(* Logix 5000 project; controller BTS01 vendor 1 type 14 code 217 rev 32.14; software revision 32.04; part 6 of 15 *)
(* tags used below, declared in another part *)
   Alarm_Active : DINT;
   Alarm_TMR : TIMER[17,32];
   ALM_ENABLE : DINT[25];
   HMI_Global_Alarm_Ack_PB : BOOL;
   HMIAlarms : DINT[25];   // Alarm Trigger Array
   HMIAlarmsMsg : STRING64[17,32];   // Alarm Descriptions to Match Alarm Trigger Array
(* Alarm, continued *)

ROUTINE Alarm_04   (* ladder *)
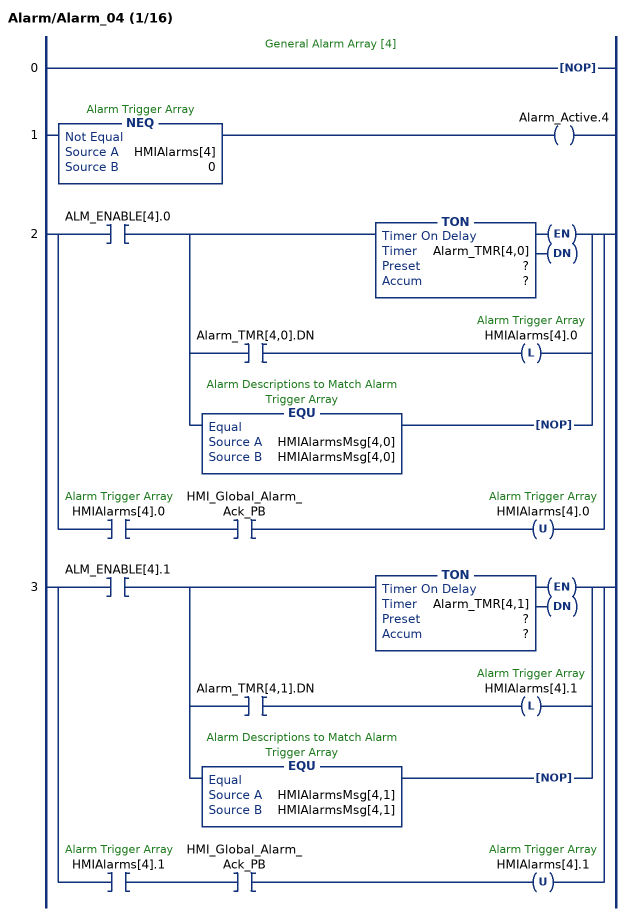
   // General Alarm Array [4]
   0: NOP();
   1: NEQ(HMIAlarms[4],0)OTE(Alarm_Active.4);
   2: [XIC(ALM_ENABLE[4].0) [TON(Alarm_TMR[4,0],?,?) ,XIC(Alarm_TMR[4,0].DN) OTL(HMIAlarms[4].0) ,EQU(HMIAlarmsMsg[4,0],HMIAlarmsMsg[4,0]) NOP() ] ,XIC(HMIAlarms[4].0) XIC(HMI_Global_Alarm_Ack_PB) OTU(HMIAlarms[4].0) ];
   3: [XIC(ALM_ENABLE[4].1) [TON(Alarm_TMR[4,1],?,?) ,XIC(Alarm_TMR[4,1].DN) OTL(HMIAlarms[4].1) ,EQU(HMIAlarmsMsg[4,1],HMIAlarmsMsg[4,1]) NOP() ] ,XIC(HMIAlarms[4].1) XIC(HMI_Global_Alarm_Ack_PB) OTU(HMIAlarms[4].1) ];
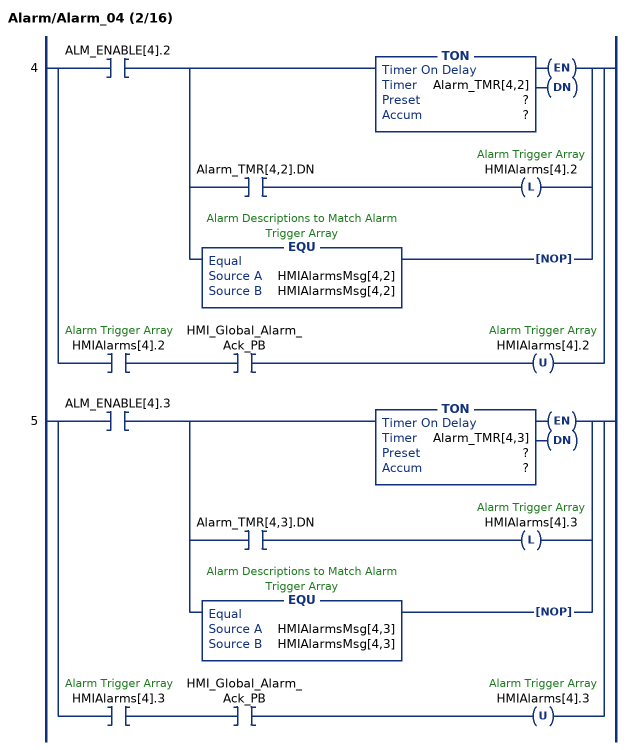
   4: [XIC(ALM_ENABLE[4].2) [TON(Alarm_TMR[4,2],?,?) ,XIC(Alarm_TMR[4,2].DN) OTL(HMIAlarms[4].2) ,EQU(HMIAlarmsMsg[4,2],HMIAlarmsMsg[4,2]) NOP() ] ,XIC(HMIAlarms[4].2) XIC(HMI_Global_Alarm_Ack_PB) OTU(HMIAlarms[4].2) ];
   5: [XIC(ALM_ENABLE[4].3) [TON(Alarm_TMR[4,3],?,?) ,XIC(Alarm_TMR[4,3].DN) OTL(HMIAlarms[4].3) ,EQU(HMIAlarmsMsg[4,3],HMIAlarmsMsg[4,3]) NOP() ] ,XIC(HMIAlarms[4].3) XIC(HMI_Global_Alarm_Ack_PB) OTU(HMIAlarms[4].3) ];
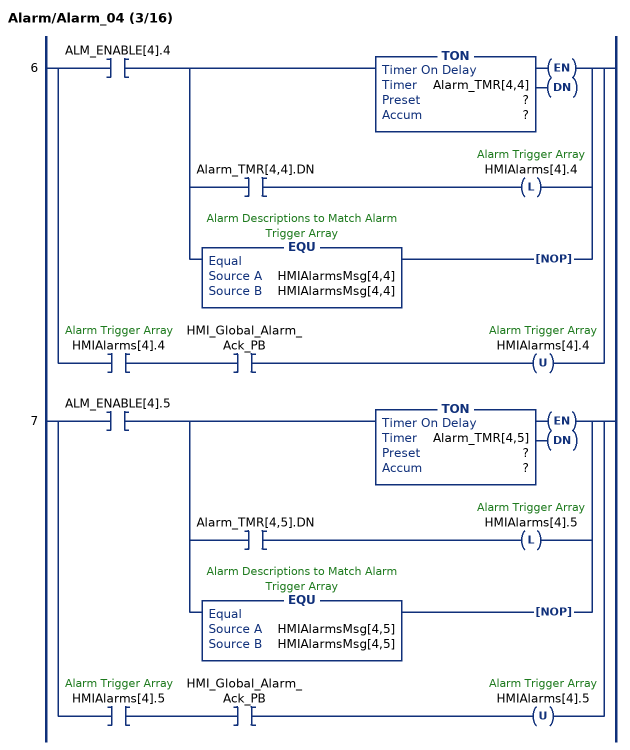
   6: [XIC(ALM_ENABLE[4].4) [TON(Alarm_TMR[4,4],?,?) ,XIC(Alarm_TMR[4,4].DN) OTL(HMIAlarms[4].4) ,EQU(HMIAlarmsMsg[4,4],HMIAlarmsMsg[4,4]) NOP() ] ,XIC(HMIAlarms[4].4) XIC(HMI_Global_Alarm_Ack_PB) OTU(HMIAlarms[4].4) ];
   7: [XIC(ALM_ENABLE[4].5) [TON(Alarm_TMR[4,5],?,?) ,XIC(Alarm_TMR[4,5].DN) OTL(HMIAlarms[4].5) ,EQU(HMIAlarmsMsg[4,5],HMIAlarmsMsg[4,5]) NOP() ] ,XIC(HMIAlarms[4].5) XIC(HMI_Global_Alarm_Ack_PB) OTU(HMIAlarms[4].5) ];
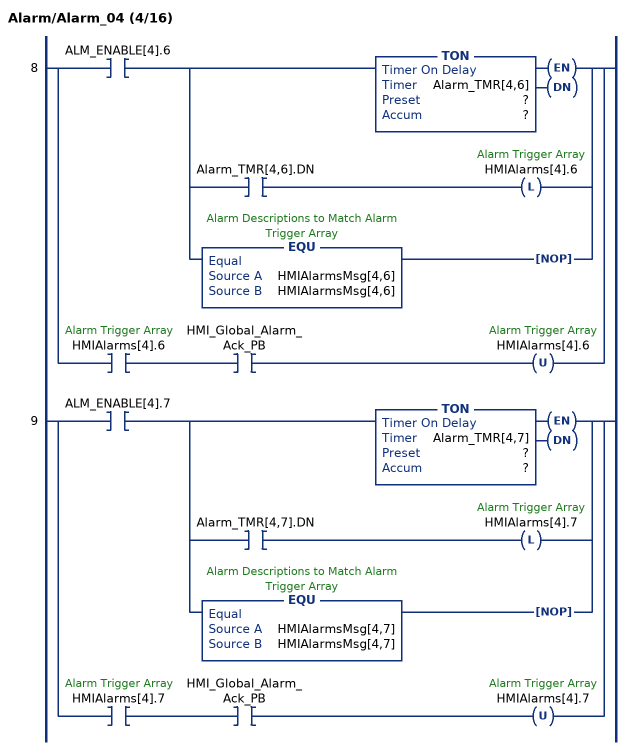
   8: [XIC(ALM_ENABLE[4].6) [TON(Alarm_TMR[4,6],?,?) ,XIC(Alarm_TMR[4,6].DN) OTL(HMIAlarms[4].6) ,EQU(HMIAlarmsMsg[4,6],HMIAlarmsMsg[4,6]) NOP() ] ,XIC(HMIAlarms[4].6) XIC(HMI_Global_Alarm_Ack_PB) OTU(HMIAlarms[4].6) ];
   9: [XIC(ALM_ENABLE[4].7) [TON(Alarm_TMR[4,7],?,?) ,XIC(Alarm_TMR[4,7].DN) OTL(HMIAlarms[4].7) ,EQU(HMIAlarmsMsg[4,7],HMIAlarmsMsg[4,7]) NOP() ] ,XIC(HMIAlarms[4].7) XIC(HMI_Global_Alarm_Ack_PB) OTU(HMIAlarms[4].7) ];
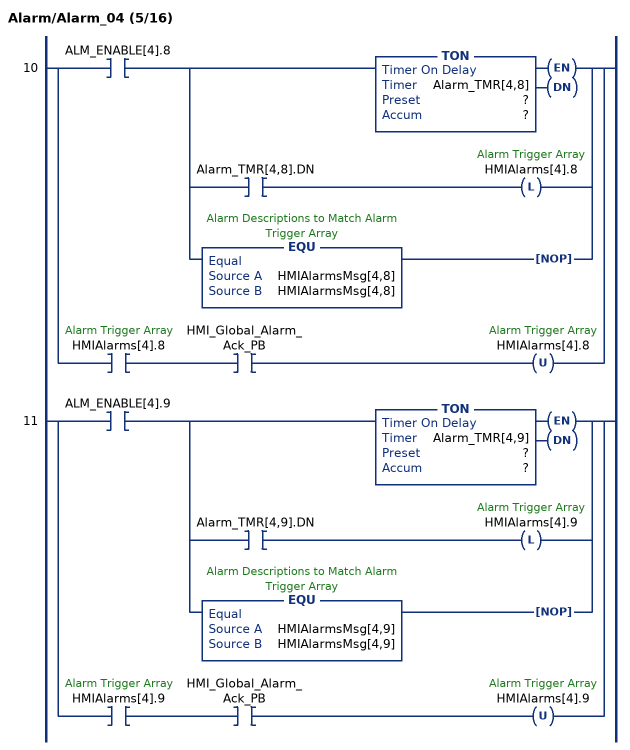
   10: [XIC(ALM_ENABLE[4].8) [TON(Alarm_TMR[4,8],?,?) ,XIC(Alarm_TMR[4,8].DN) OTL(HMIAlarms[4].8) ,EQU(HMIAlarmsMsg[4,8],HMIAlarmsMsg[4,8]) NOP() ] ,XIC(HMIAlarms[4].8) XIC(HMI_Global_Alarm_Ack_PB) OTU(HMIAlarms[4].8) ];
   11: [XIC(ALM_ENABLE[4].9) [TON(Alarm_TMR[4,9],?,?) ,XIC(Alarm_TMR[4,9].DN) OTL(HMIAlarms[4].9) ,EQU(HMIAlarmsMsg[4,9],HMIAlarmsMsg[4,9]) NOP() ] ,XIC(HMIAlarms[4].9) XIC(HMI_Global_Alarm_Ack_PB) OTU(HMIAlarms[4].9) ];
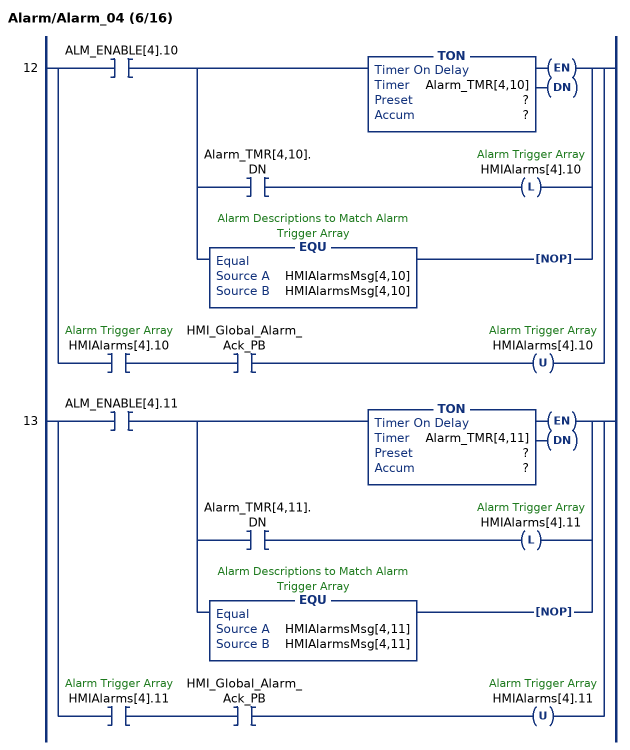
   12: [XIC(ALM_ENABLE[4].10) [TON(Alarm_TMR[4,10],?,?) ,XIC(Alarm_TMR[4,10].DN) OTL(HMIAlarms[4].10) ,EQU(HMIAlarmsMsg[4,10],HMIAlarmsMsg[4,10]) NOP() ] ,XIC(HMIAlarms[4].10) XIC(HMI_Global_Alarm_Ack_PB) OTU(HMIAlarms[4].10) ];
   13: [XIC(ALM_ENABLE[4].11) [TON(Alarm_TMR[4,11],?,?) ,XIC(Alarm_TMR[4,11].DN) OTL(HMIAlarms[4].11) ,EQU(HMIAlarmsMsg[4,11],HMIAlarmsMsg[4,11]) NOP() ] ,XIC(HMIAlarms[4].11) XIC(HMI_Global_Alarm_Ack_PB) OTU(HMIAlarms[4].11) ];
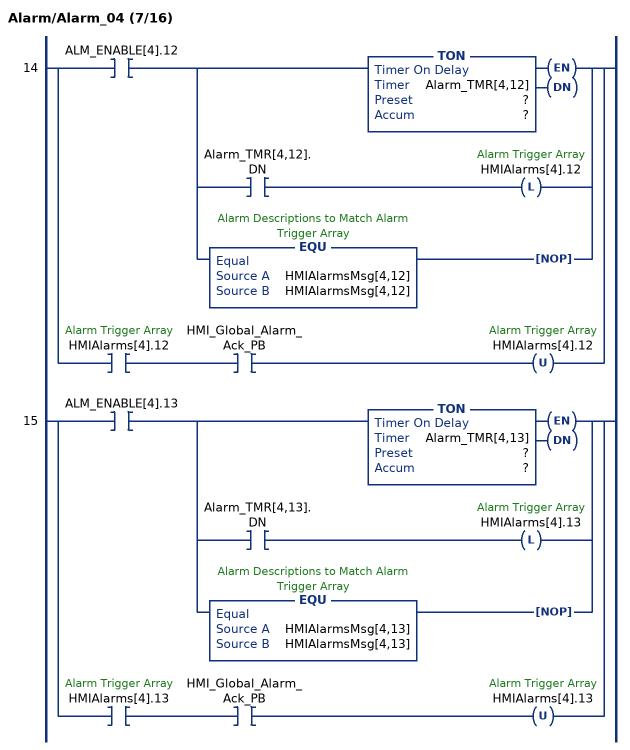
   14: [XIC(ALM_ENABLE[4].12) [TON(Alarm_TMR[4,12],?,?) ,XIC(Alarm_TMR[4,12].DN) OTL(HMIAlarms[4].12) ,EQU(HMIAlarmsMsg[4,12],HMIAlarmsMsg[4,12]) NOP() ] ,XIC(HMIAlarms[4].12) XIC(HMI_Global_Alarm_Ack_PB) OTU(HMIAlarms[4].12) ];
   15: [XIC(ALM_ENABLE[4].13) [TON(Alarm_TMR[4,13],?,?) ,XIC(Alarm_TMR[4,13].DN) OTL(HMIAlarms[4].13) ,EQU(HMIAlarmsMsg[4,13],HMIAlarmsMsg[4,13]) NOP() ] ,XIC(HMIAlarms[4].13) XIC(HMI_Global_Alarm_Ack_PB) OTU(HMIAlarms[4].13) ];
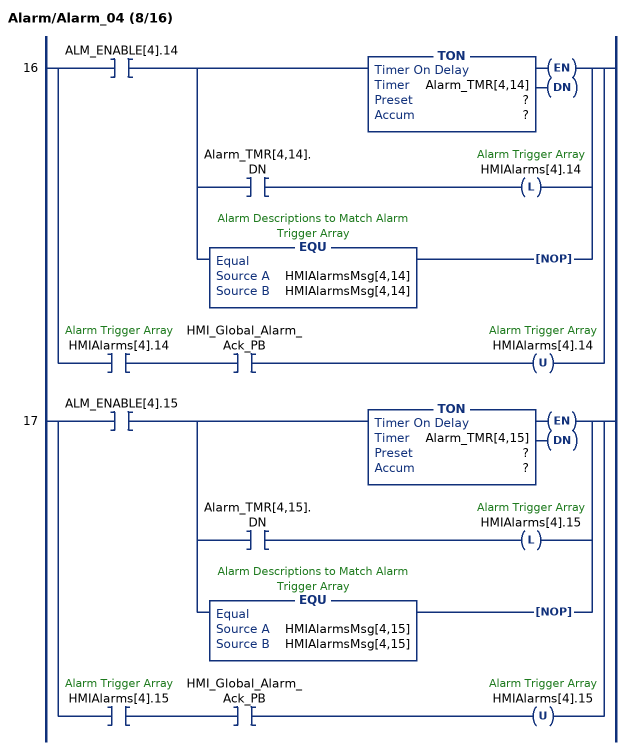
   16: [XIC(ALM_ENABLE[4].14) [TON(Alarm_TMR[4,14],?,?) ,XIC(Alarm_TMR[4,14].DN) OTL(HMIAlarms[4].14) ,EQU(HMIAlarmsMsg[4,14],HMIAlarmsMsg[4,14]) NOP() ] ,XIC(HMIAlarms[4].14) XIC(HMI_Global_Alarm_Ack_PB) OTU(HMIAlarms[4].14) ];
   17: [XIC(ALM_ENABLE[4].15) [TON(Alarm_TMR[4,15],?,?) ,XIC(Alarm_TMR[4,15].DN) OTL(HMIAlarms[4].15) ,EQU(HMIAlarmsMsg[4,15],HMIAlarmsMsg[4,15]) NOP() ] ,XIC(HMIAlarms[4].15) XIC(HMI_Global_Alarm_Ack_PB) OTU(HMIAlarms[4].15) ];
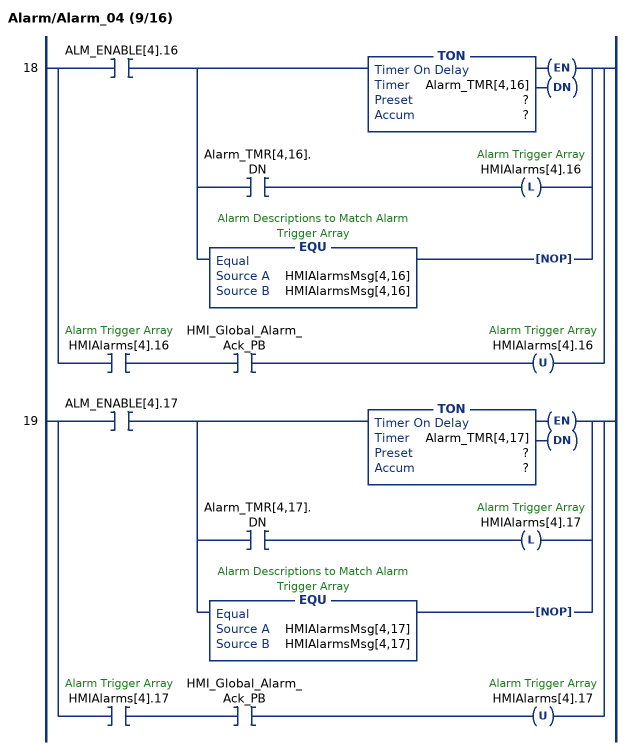
   18: [XIC(ALM_ENABLE[4].16) [TON(Alarm_TMR[4,16],?,?) ,XIC(Alarm_TMR[4,16].DN) OTL(HMIAlarms[4].16) ,EQU(HMIAlarmsMsg[4,16],HMIAlarmsMsg[4,16]) NOP() ] ,XIC(HMIAlarms[4].16) XIC(HMI_Global_Alarm_Ack_PB) OTU(HMIAlarms[4].16) ];
   19: [XIC(ALM_ENABLE[4].17) [TON(Alarm_TMR[4,17],?,?) ,XIC(Alarm_TMR[4,17].DN) OTL(HMIAlarms[4].17) ,EQU(HMIAlarmsMsg[4,17],HMIAlarmsMsg[4,17]) NOP() ] ,XIC(HMIAlarms[4].17) XIC(HMI_Global_Alarm_Ack_PB) OTU(HMIAlarms[4].17) ];
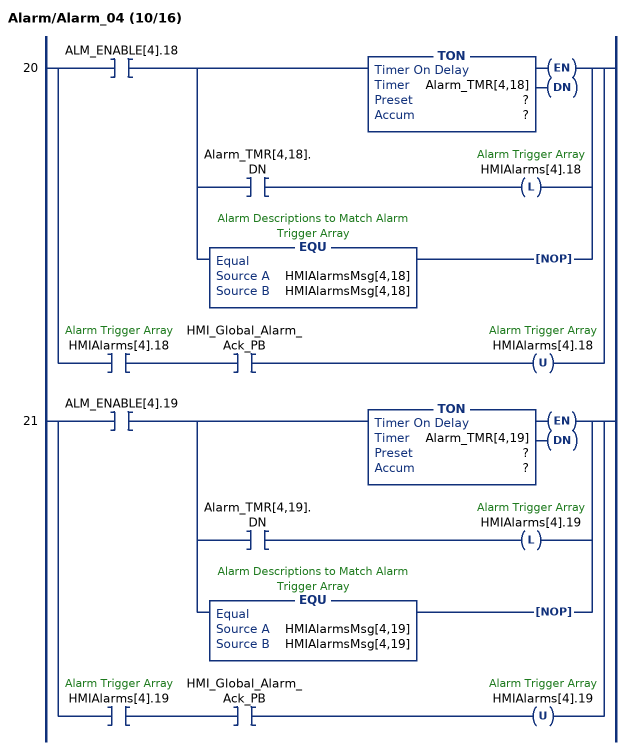
   20: [XIC(ALM_ENABLE[4].18) [TON(Alarm_TMR[4,18],?,?) ,XIC(Alarm_TMR[4,18].DN) OTL(HMIAlarms[4].18) ,EQU(HMIAlarmsMsg[4,18],HMIAlarmsMsg[4,18]) NOP() ] ,XIC(HMIAlarms[4].18) XIC(HMI_Global_Alarm_Ack_PB) OTU(HMIAlarms[4].18) ];
   21: [XIC(ALM_ENABLE[4].19) [TON(Alarm_TMR[4,19],?,?) ,XIC(Alarm_TMR[4,19].DN) OTL(HMIAlarms[4].19) ,EQU(HMIAlarmsMsg[4,19],HMIAlarmsMsg[4,19]) NOP() ] ,XIC(HMIAlarms[4].19) XIC(HMI_Global_Alarm_Ack_PB) OTU(HMIAlarms[4].19) ];
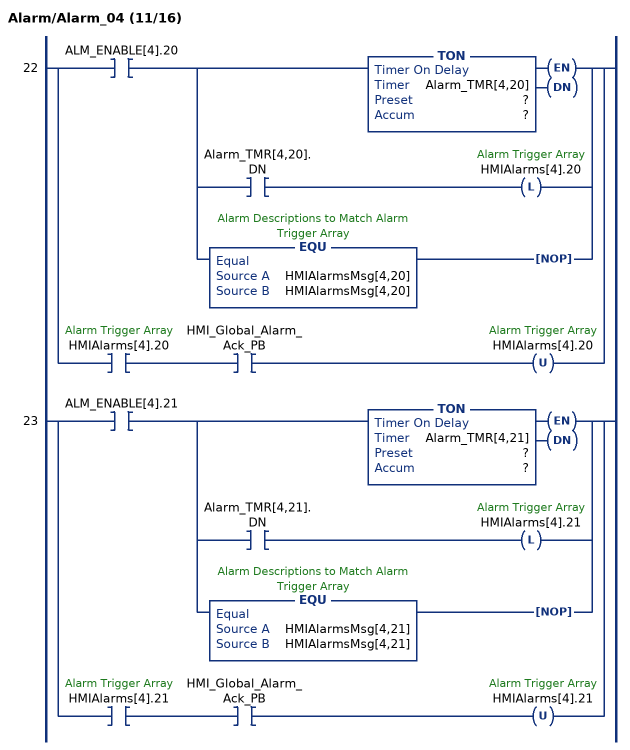
   22: [XIC(ALM_ENABLE[4].20) [TON(Alarm_TMR[4,20],?,?) ,XIC(Alarm_TMR[4,20].DN) OTL(HMIAlarms[4].20) ,EQU(HMIAlarmsMsg[4,20],HMIAlarmsMsg[4,20]) NOP() ] ,XIC(HMIAlarms[4].20) XIC(HMI_Global_Alarm_Ack_PB) OTU(HMIAlarms[4].20) ];
   23: [XIC(ALM_ENABLE[4].21) [TON(Alarm_TMR[4,21],?,?) ,XIC(Alarm_TMR[4,21].DN) OTL(HMIAlarms[4].21) ,EQU(HMIAlarmsMsg[4,21],HMIAlarmsMsg[4,21]) NOP() ] ,XIC(HMIAlarms[4].21) XIC(HMI_Global_Alarm_Ack_PB) OTU(HMIAlarms[4].21) ];
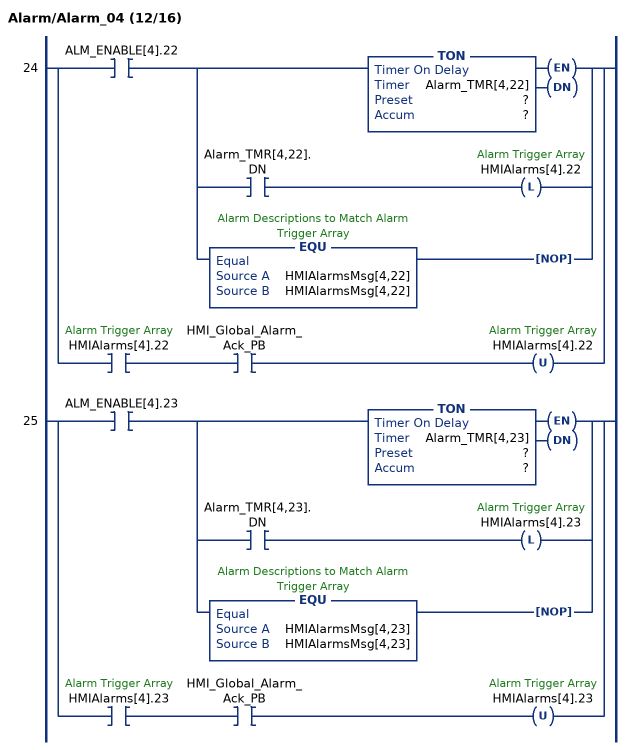
   24: [XIC(ALM_ENABLE[4].22) [TON(Alarm_TMR[4,22],?,?) ,XIC(Alarm_TMR[4,22].DN) OTL(HMIAlarms[4].22) ,EQU(HMIAlarmsMsg[4,22],HMIAlarmsMsg[4,22]) NOP() ] ,XIC(HMIAlarms[4].22) XIC(HMI_Global_Alarm_Ack_PB) OTU(HMIAlarms[4].22) ];
   25: [XIC(ALM_ENABLE[4].23) [TON(Alarm_TMR[4,23],?,?) ,XIC(Alarm_TMR[4,23].DN) OTL(HMIAlarms[4].23) ,EQU(HMIAlarmsMsg[4,23],HMIAlarmsMsg[4,23]) NOP() ] ,XIC(HMIAlarms[4].23) XIC(HMI_Global_Alarm_Ack_PB) OTU(HMIAlarms[4].23) ];
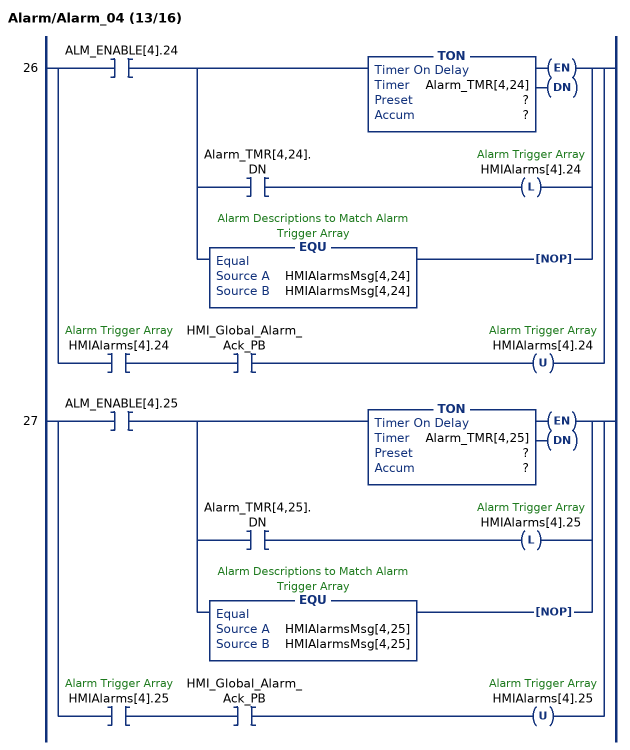
   26: [XIC(ALM_ENABLE[4].24) [TON(Alarm_TMR[4,24],?,?) ,XIC(Alarm_TMR[4,24].DN) OTL(HMIAlarms[4].24) ,EQU(HMIAlarmsMsg[4,24],HMIAlarmsMsg[4,24]) NOP() ] ,XIC(HMIAlarms[4].24) XIC(HMI_Global_Alarm_Ack_PB) OTU(HMIAlarms[4].24) ];
   27: [XIC(ALM_ENABLE[4].25) [TON(Alarm_TMR[4,25],?,?) ,XIC(Alarm_TMR[4,25].DN) OTL(HMIAlarms[4].25) ,EQU(HMIAlarmsMsg[4,25],HMIAlarmsMsg[4,25]) NOP() ] ,XIC(HMIAlarms[4].25) XIC(HMI_Global_Alarm_Ack_PB) OTU(HMIAlarms[4].25) ];
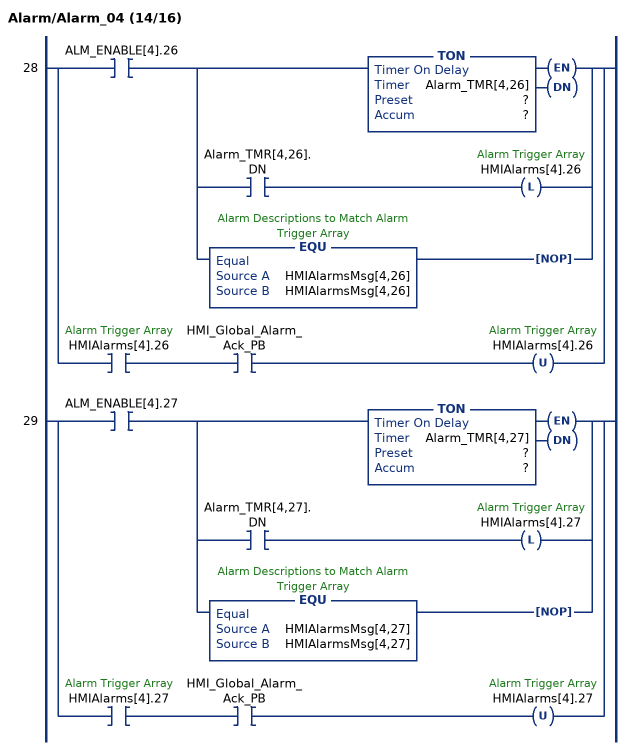
   28: [XIC(ALM_ENABLE[4].26) [TON(Alarm_TMR[4,26],?,?) ,XIC(Alarm_TMR[4,26].DN) OTL(HMIAlarms[4].26) ,EQU(HMIAlarmsMsg[4,26],HMIAlarmsMsg[4,26]) NOP() ] ,XIC(HMIAlarms[4].26) XIC(HMI_Global_Alarm_Ack_PB) OTU(HMIAlarms[4].26) ];
   29: [XIC(ALM_ENABLE[4].27) [TON(Alarm_TMR[4,27],?,?) ,XIC(Alarm_TMR[4,27].DN) OTL(HMIAlarms[4].27) ,EQU(HMIAlarmsMsg[4,27],HMIAlarmsMsg[4,27]) NOP() ] ,XIC(HMIAlarms[4].27) XIC(HMI_Global_Alarm_Ack_PB) OTU(HMIAlarms[4].27) ];
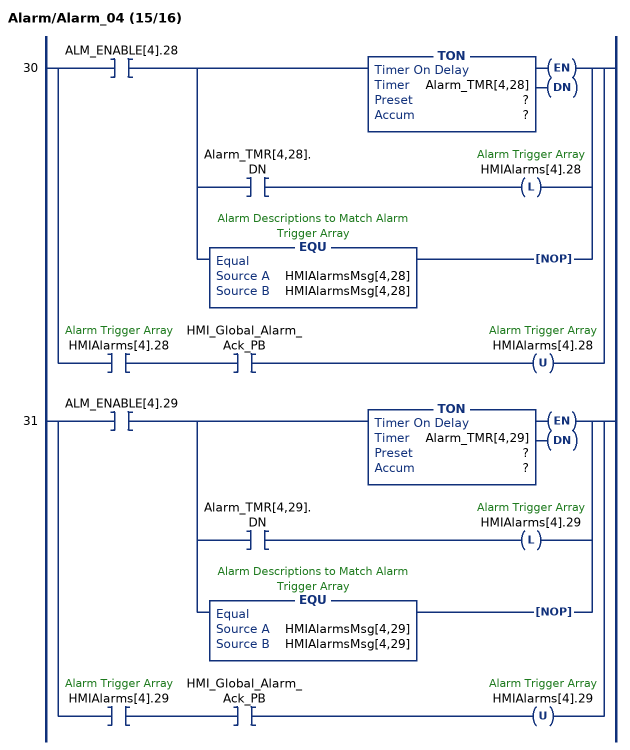
   30: [XIC(ALM_ENABLE[4].28) [TON(Alarm_TMR[4,28],?,?) ,XIC(Alarm_TMR[4,28].DN) OTL(HMIAlarms[4].28) ,EQU(HMIAlarmsMsg[4,28],HMIAlarmsMsg[4,28]) NOP() ] ,XIC(HMIAlarms[4].28) XIC(HMI_Global_Alarm_Ack_PB) OTU(HMIAlarms[4].28) ];
   31: [XIC(ALM_ENABLE[4].29) [TON(Alarm_TMR[4,29],?,?) ,XIC(Alarm_TMR[4,29].DN) OTL(HMIAlarms[4].29) ,EQU(HMIAlarmsMsg[4,29],HMIAlarmsMsg[4,29]) NOP() ] ,XIC(HMIAlarms[4].29) XIC(HMI_Global_Alarm_Ack_PB) OTU(HMIAlarms[4].29) ];
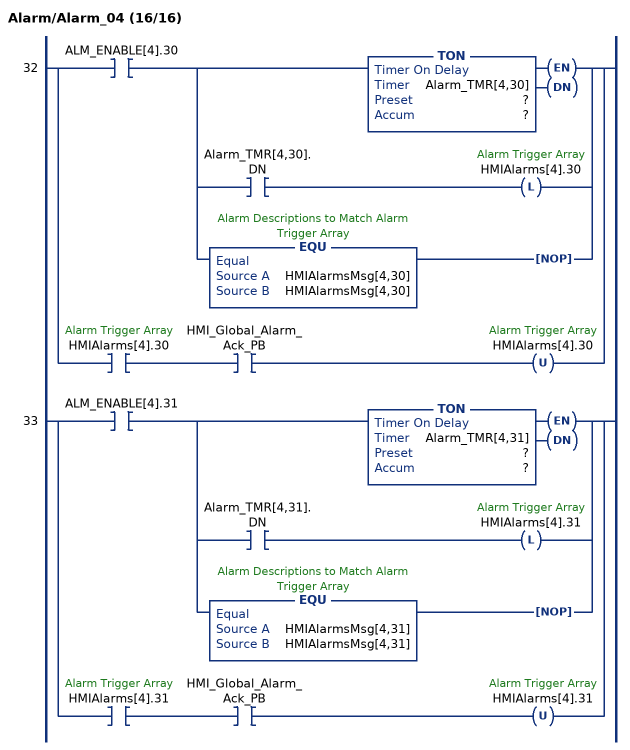
   32: [XIC(ALM_ENABLE[4].30) [TON(Alarm_TMR[4,30],?,?) ,XIC(Alarm_TMR[4,30].DN) OTL(HMIAlarms[4].30) ,EQU(HMIAlarmsMsg[4,30],HMIAlarmsMsg[4,30]) NOP() ] ,XIC(HMIAlarms[4].30) XIC(HMI_Global_Alarm_Ack_PB) OTU(HMIAlarms[4].30) ];
   33: [XIC(ALM_ENABLE[4].31) [TON(Alarm_TMR[4,31],?,?) ,XIC(Alarm_TMR[4,31].DN) OTL(HMIAlarms[4].31) ,EQU(HMIAlarmsMsg[4,31],HMIAlarmsMsg[4,31]) NOP() ] ,XIC(HMIAlarms[4].31) XIC(HMI_Global_Alarm_Ack_PB) OTU(HMIAlarms[4].31) ];
END_ROUTINE

ROUTINE Alarm_05   (* ladder *)
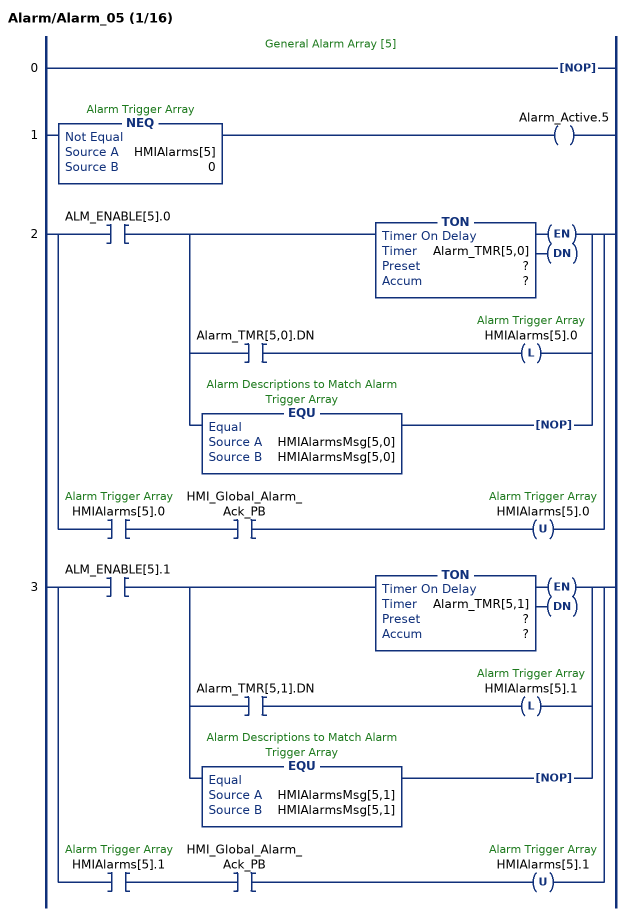
   // General Alarm Array [5]
   0: NOP();
   1: NEQ(HMIAlarms[5],0)OTE(Alarm_Active.5);
   2: [XIC(ALM_ENABLE[5].0) [TON(Alarm_TMR[5,0],?,?) ,XIC(Alarm_TMR[5,0].DN) OTL(HMIAlarms[5].0) ,EQU(HMIAlarmsMsg[5,0],HMIAlarmsMsg[5,0]) NOP() ] ,XIC(HMIAlarms[5].0) XIC(HMI_Global_Alarm_Ack_PB) OTU(HMIAlarms[5].0) ];
   3: [XIC(ALM_ENABLE[5].1) [TON(Alarm_TMR[5,1],?,?) ,XIC(Alarm_TMR[5,1].DN) OTL(HMIAlarms[5].1) ,EQU(HMIAlarmsMsg[5,1],HMIAlarmsMsg[5,1]) NOP() ] ,XIC(HMIAlarms[5].1) XIC(HMI_Global_Alarm_Ack_PB) OTU(HMIAlarms[5].1) ];
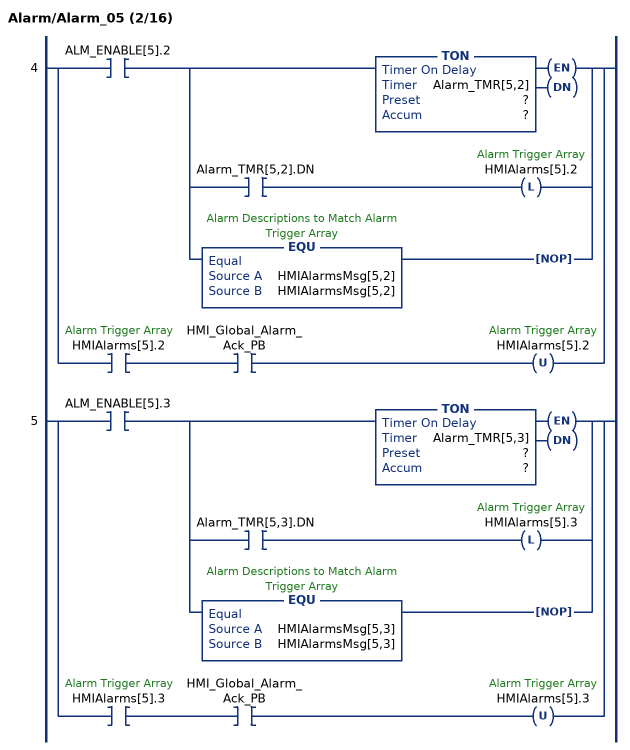
   4: [XIC(ALM_ENABLE[5].2) [TON(Alarm_TMR[5,2],?,?) ,XIC(Alarm_TMR[5,2].DN) OTL(HMIAlarms[5].2) ,EQU(HMIAlarmsMsg[5,2],HMIAlarmsMsg[5,2]) NOP() ] ,XIC(HMIAlarms[5].2) XIC(HMI_Global_Alarm_Ack_PB) OTU(HMIAlarms[5].2) ];
   5: [XIC(ALM_ENABLE[5].3) [TON(Alarm_TMR[5,3],?,?) ,XIC(Alarm_TMR[5,3].DN) OTL(HMIAlarms[5].3) ,EQU(HMIAlarmsMsg[5,3],HMIAlarmsMsg[5,3]) NOP() ] ,XIC(HMIAlarms[5].3) XIC(HMI_Global_Alarm_Ack_PB) OTU(HMIAlarms[5].3) ];
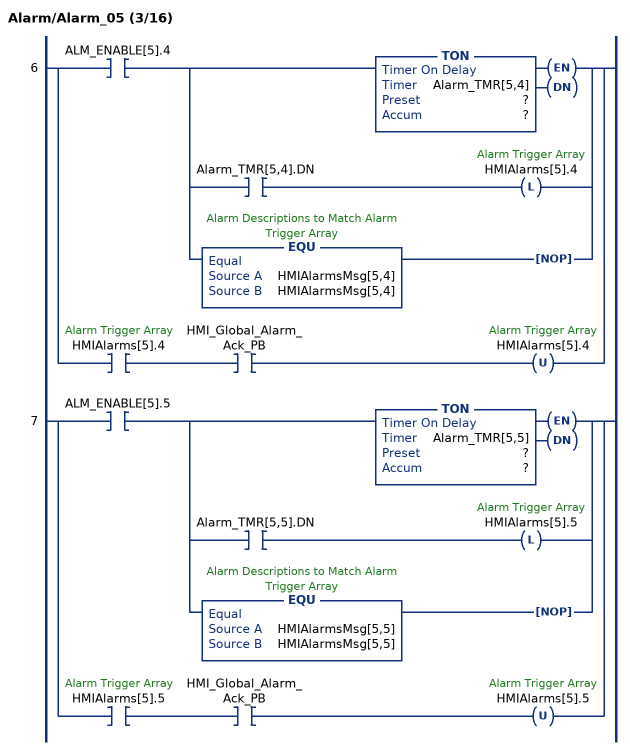
   6: [XIC(ALM_ENABLE[5].4) [TON(Alarm_TMR[5,4],?,?) ,XIC(Alarm_TMR[5,4].DN) OTL(HMIAlarms[5].4) ,EQU(HMIAlarmsMsg[5,4],HMIAlarmsMsg[5,4]) NOP() ] ,XIC(HMIAlarms[5].4) XIC(HMI_Global_Alarm_Ack_PB) OTU(HMIAlarms[5].4) ];
   7: [XIC(ALM_ENABLE[5].5) [TON(Alarm_TMR[5,5],?,?) ,XIC(Alarm_TMR[5,5].DN) OTL(HMIAlarms[5].5) ,EQU(HMIAlarmsMsg[5,5],HMIAlarmsMsg[5,5]) NOP() ] ,XIC(HMIAlarms[5].5) XIC(HMI_Global_Alarm_Ack_PB) OTU(HMIAlarms[5].5) ];
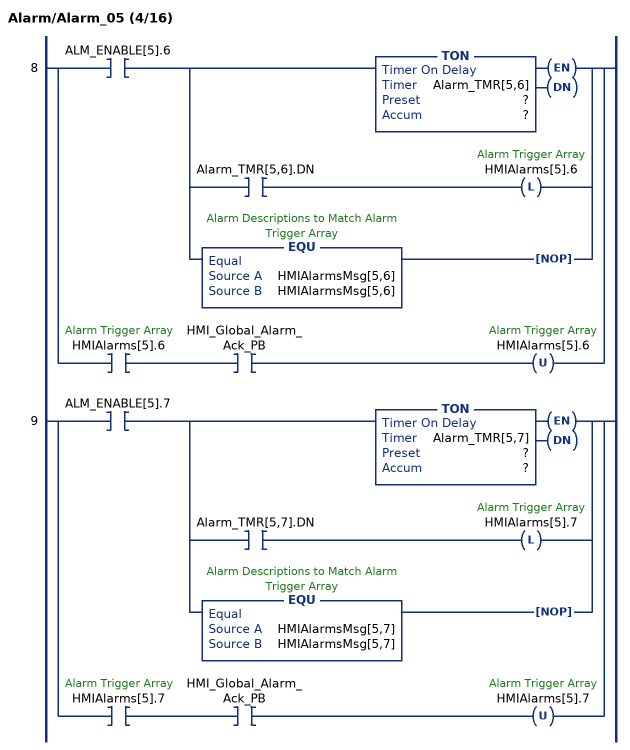
   8: [XIC(ALM_ENABLE[5].6) [TON(Alarm_TMR[5,6],?,?) ,XIC(Alarm_TMR[5,6].DN) OTL(HMIAlarms[5].6) ,EQU(HMIAlarmsMsg[5,6],HMIAlarmsMsg[5,6]) NOP() ] ,XIC(HMIAlarms[5].6) XIC(HMI_Global_Alarm_Ack_PB) OTU(HMIAlarms[5].6) ];
   9: [XIC(ALM_ENABLE[5].7) [TON(Alarm_TMR[5,7],?,?) ,XIC(Alarm_TMR[5,7].DN) OTL(HMIAlarms[5].7) ,EQU(HMIAlarmsMsg[5,7],HMIAlarmsMsg[5,7]) NOP() ] ,XIC(HMIAlarms[5].7) XIC(HMI_Global_Alarm_Ack_PB) OTU(HMIAlarms[5].7) ];
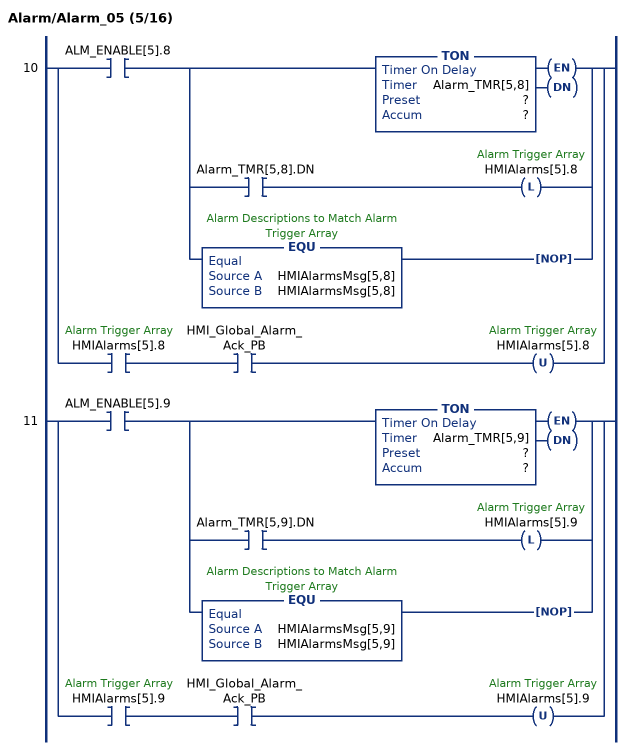
   10: [XIC(ALM_ENABLE[5].8) [TON(Alarm_TMR[5,8],?,?) ,XIC(Alarm_TMR[5,8].DN) OTL(HMIAlarms[5].8) ,EQU(HMIAlarmsMsg[5,8],HMIAlarmsMsg[5,8]) NOP() ] ,XIC(HMIAlarms[5].8) XIC(HMI_Global_Alarm_Ack_PB) OTU(HMIAlarms[5].8) ];
   11: [XIC(ALM_ENABLE[5].9) [TON(Alarm_TMR[5,9],?,?) ,XIC(Alarm_TMR[5,9].DN) OTL(HMIAlarms[5].9) ,EQU(HMIAlarmsMsg[5,9],HMIAlarmsMsg[5,9]) NOP() ] ,XIC(HMIAlarms[5].9) XIC(HMI_Global_Alarm_Ack_PB) OTU(HMIAlarms[5].9) ];
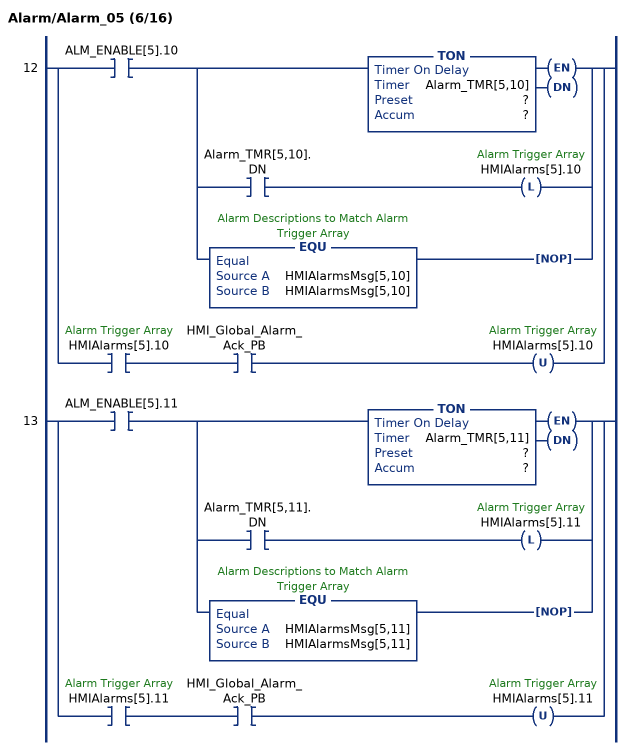
   12: [XIC(ALM_ENABLE[5].10) [TON(Alarm_TMR[5,10],?,?) ,XIC(Alarm_TMR[5,10].DN) OTL(HMIAlarms[5].10) ,EQU(HMIAlarmsMsg[5,10],HMIAlarmsMsg[5,10]) NOP() ] ,XIC(HMIAlarms[5].10) XIC(HMI_Global_Alarm_Ack_PB) OTU(HMIAlarms[5].10) ];
   13: [XIC(ALM_ENABLE[5].11) [TON(Alarm_TMR[5,11],?,?) ,XIC(Alarm_TMR[5,11].DN) OTL(HMIAlarms[5].11) ,EQU(HMIAlarmsMsg[5,11],HMIAlarmsMsg[5,11]) NOP() ] ,XIC(HMIAlarms[5].11) XIC(HMI_Global_Alarm_Ack_PB) OTU(HMIAlarms[5].11) ];
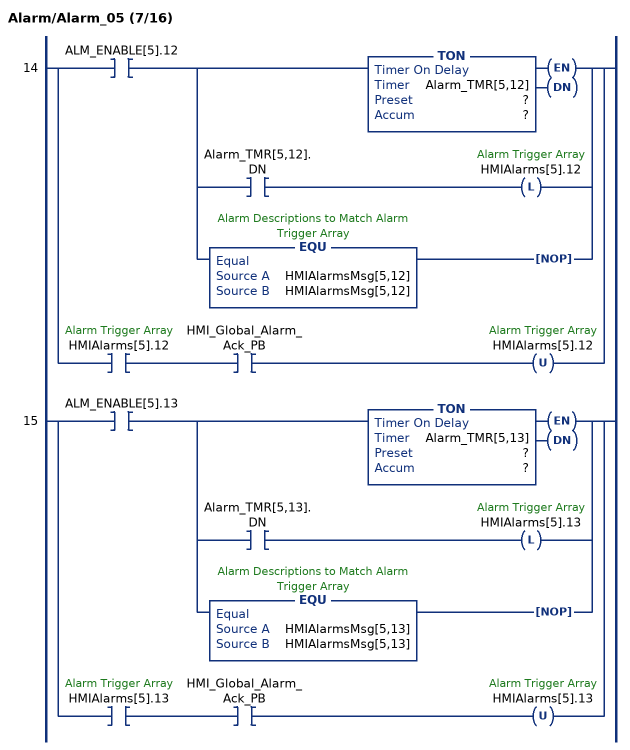
   14: [XIC(ALM_ENABLE[5].12) [TON(Alarm_TMR[5,12],?,?) ,XIC(Alarm_TMR[5,12].DN) OTL(HMIAlarms[5].12) ,EQU(HMIAlarmsMsg[5,12],HMIAlarmsMsg[5,12]) NOP() ] ,XIC(HMIAlarms[5].12) XIC(HMI_Global_Alarm_Ack_PB) OTU(HMIAlarms[5].12) ];
   15: [XIC(ALM_ENABLE[5].13) [TON(Alarm_TMR[5,13],?,?) ,XIC(Alarm_TMR[5,13].DN) OTL(HMIAlarms[5].13) ,EQU(HMIAlarmsMsg[5,13],HMIAlarmsMsg[5,13]) NOP() ] ,XIC(HMIAlarms[5].13) XIC(HMI_Global_Alarm_Ack_PB) OTU(HMIAlarms[5].13) ];
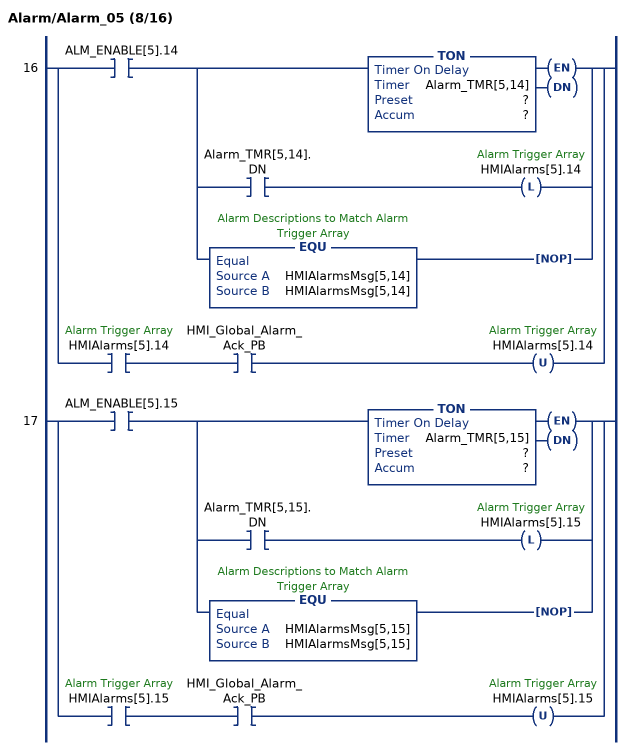
   16: [XIC(ALM_ENABLE[5].14) [TON(Alarm_TMR[5,14],?,?) ,XIC(Alarm_TMR[5,14].DN) OTL(HMIAlarms[5].14) ,EQU(HMIAlarmsMsg[5,14],HMIAlarmsMsg[5,14]) NOP() ] ,XIC(HMIAlarms[5].14) XIC(HMI_Global_Alarm_Ack_PB) OTU(HMIAlarms[5].14) ];
   17: [XIC(ALM_ENABLE[5].15) [TON(Alarm_TMR[5,15],?,?) ,XIC(Alarm_TMR[5,15].DN) OTL(HMIAlarms[5].15) ,EQU(HMIAlarmsMsg[5,15],HMIAlarmsMsg[5,15]) NOP() ] ,XIC(HMIAlarms[5].15) XIC(HMI_Global_Alarm_Ack_PB) OTU(HMIAlarms[5].15) ];
